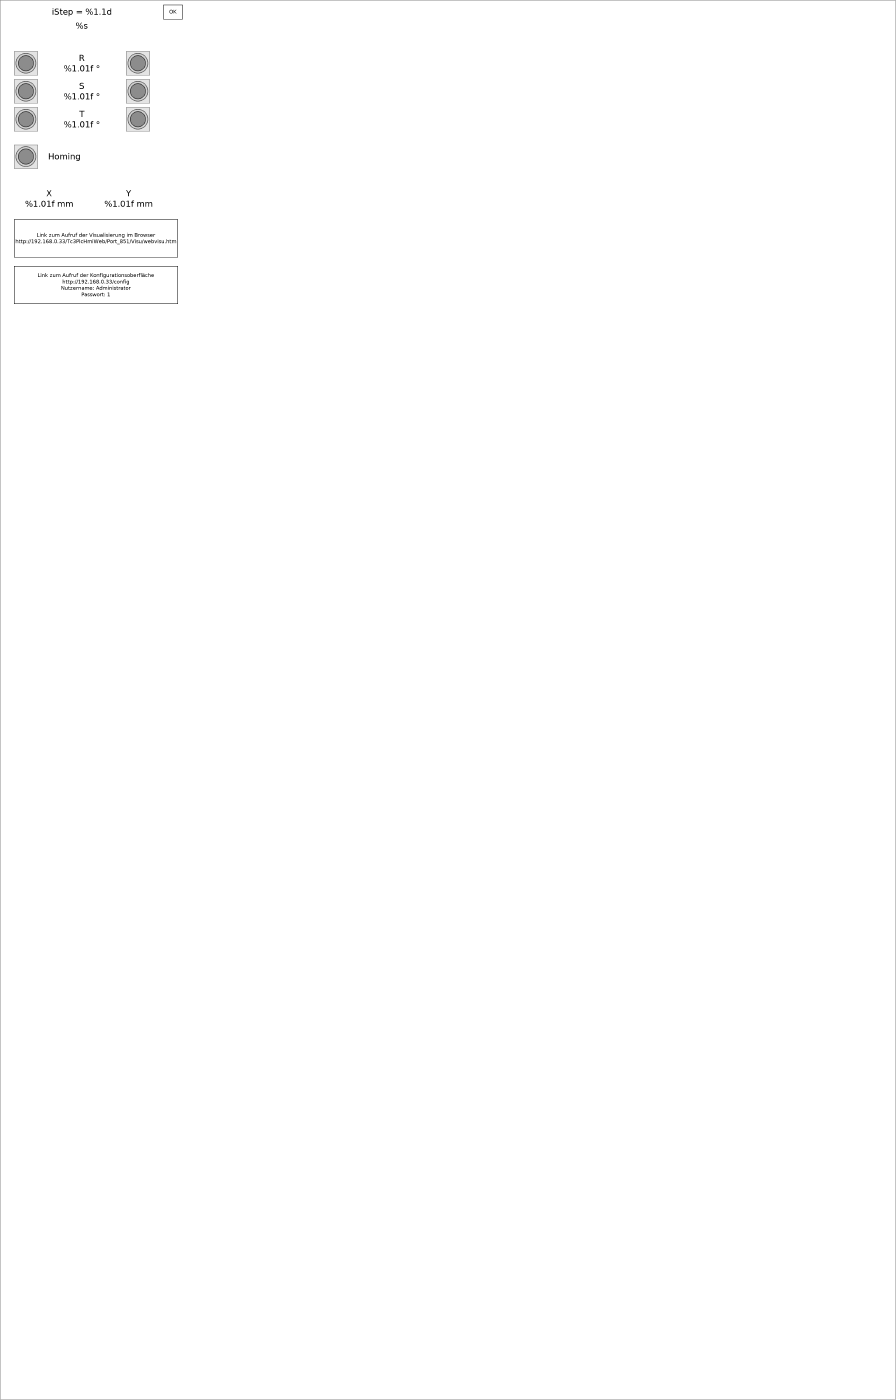
VISUALIZATION Visualization  // 1920x3000
    Rectangle (30,470 351x81), "Link zum Aufruf der Visualisierung im Browser http://192.168.0.33/Tc3PlcHmiWeb/Port_851/Visu/webvisu.htm"
    PushSwitch (270,110 51x51), variable: MC.bRstepP, behaviour: TAP, style: Switch-PushSwitch-Gray
    PushSwitch (30,110 51x51), variable: MC.bRstepM, behaviour: TAP, style: Switch-PushSwitch-Gray
    PushSwitch (30,310 51x51), variable: MC.bHoming, behaviour: TAP, style: Switch-PushSwitch-Gray
    Label (100,310 91x51), "Homing"
    Rectangle (90,110 171x51), "R %1.01f °", text variable: MC.ax_r.dActPos
    Rectangle (10,10 331x31), "iStep = %1.1d", text variable: MC.iStep
    Rectangle (10,40 331x31), "%s", text variable: MC.sStep
    Rectangle (350,10 41x31), "OK"
        tap MC.bOk
    PushSwitch (270,170 51x51), variable: MC.bSstepP, behaviour: TAP, style: Switch-PushSwitch-Gray
    PushSwitch (30,170 51x51), variable: MC.bSstepM, behaviour: TAP, style: Switch-PushSwitch-Gray
    Rectangle (90,170 171x51), "S %1.01f °", text variable: MC.ax_s.dActPos
    PushSwitch (270,230 51x51), variable: MC.bTstepP, behaviour: TAP, style: Switch-PushSwitch-Gray
    PushSwitch (30,230 51x51), variable: MC.bTstepM, behaviour: TAP, style: Switch-PushSwitch-Gray
    Rectangle (90,230 171x51), "T %1.01f °", text variable: MC.ax_t.dActPos
    Rectangle (20,400 171x51), "X %1.01f mm", text variable: MC.touch_scale_x.rX_mm
    Rectangle (190,400 171x51), "Y %1.01f mm", text variable: MC.touch_scale_y.rX_mm
    Rectangle (30,570 351x81), "Link zum Aufruf der Konfigurationsoberfläche http://192.168.0.33/config Nutzername: Administrator Passwort: 1"
END_VISUALIZATION

(* stored: Version 1.1.0.1, ProductVersion 3.1.4024.6
   Visu Visualization: Id {4c19cea1-475c-4ab7-8047-42bdc9d69985} *)
